FUNCTION_BLOCK FB_PlantControl_B28

VAR
	Plant_Control : PlantAndCMs.FB_PlantControl_V2;
	
	
	MB_START : BOOL;
	MB_EMG_STOP : BOOL;
END_VAR

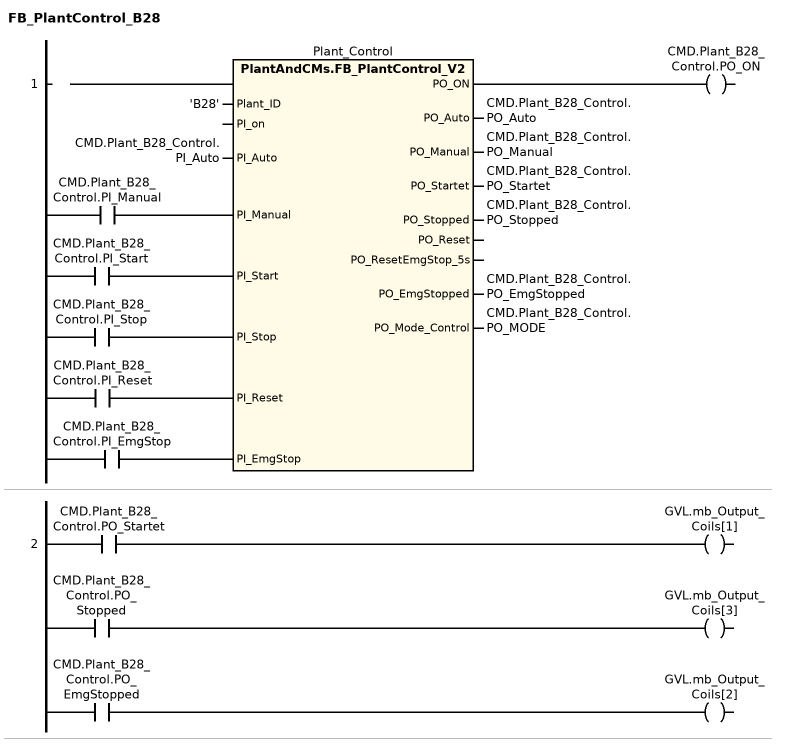
// NETWORK 1
Plant_Control(
    Plant_ID := 'B28',
    PI_Auto := CMD.Plant_B28_Control.PI_Auto,
    PI_Manual := CMD.Plant_B28_Control.PI_Manual,
    PI_Start := CMD.Plant_B28_Control.PI_Start,
    PI_Stop := CMD.Plant_B28_Control.PI_Stop,
    PI_Reset := CMD.Plant_B28_Control.PI_Reset,
    PI_EmgStop := CMD.Plant_B28_Control.PI_EmgStop,
    PO_Auto => CMD.Plant_B28_Control.PO_Auto,
    PO_Manual => CMD.Plant_B28_Control.PO_Manual,
    PO_Startet => CMD.Plant_B28_Control.PO_Startet,
    PO_Stopped => CMD.Plant_B28_Control.PO_Stopped,
    PO_EmgStopped => CMD.Plant_B28_Control.PO_EmgStopped,
    PO_Mode_Control => CMD.Plant_B28_Control.PO_MODE); // PlantAndCMs.FB_PlantControl_V2
CMD.Plant_B28_Control.PO_ON := Plant_Control.PO_ON;

// NETWORK 2
GVL.mb_Output_Coils[1] := CMD.Plant_B28_Control.PO_Startet;
GVL.mb_Output_Coils[3] := CMD.Plant_B28_Control.PO_Stopped;
GVL.mb_Output_Coils[2] := CMD.Plant_B28_Control.PO_EmgStopped;

END_FUNCTION_BLOCK

(* stored: Version 1.1.0.1, ProductVersion 3.1.4024.13
   POU FB_PlantControl_B28: Id {51d3ca2e-f57b-43c9-a2f4-cc6963402968}, SpecialFunc None *)
